// TIA Portal V16 export
// export: Created 2021-04-06T19:52:18.3847886Z, ExportSetting WithDefaults, DisplayName Totally Integrated Automation Portal, DisplayVersion V16, DisplayName TIA Portal Version Control Interface, DisplayVersion V16, DisplayName TIA Portal Openness, DisplayVersion V16, DisplayName STEP 7 Professional, DisplayVersion V16, DisplayName STEP 7 Safety, DisplayVersion V16, DisplayName WinCC Unified SCADA Engineering System, DisplayVersion V16
VAR_GLOBAL   // PLC tag table "input"
   buttonControlCircuit AT %I0.0 : Bool;   // цепи управления
   buttonStart AT %I0.1 : Bool;   // Старт
   buttonStop AT %I0.2 : Bool;   // Стоп
   buttonAlarmStop AT %I0.3 : Bool;   // Аварийный стоп
   M1_alarmCB AT %I0.4 : Bool;   // М1 - авария автоматического выключателя
   M2_alarmCB AT %I0.5 : Bool;   // М2 - авария автоматического выключателя
   isNormalElectrical AT %I0.6 : Bool;   // Сеть в норме
   sensorOverflowReceiverTable AT %I0.7 : Bool;   // Датчик пересыпа приемного стола
   YP1_ReadyAccept AT %I1.0 : Bool;   // УП1 - готов принять
   YP1_StartDozing AT %I1.1 : Bool;   // УП1 - запуск дозирования
   YP2_ReadyAccept AT %I1.2 : Bool;   // УП2 - готов принять
   YP2_StartDozing AT %I1.3 : Bool;   // УП2 - запуск дозирования
END_VAR
